Fanuc TP program (LS listing): both_features.ls

/PROG  BOTH_TEST
/ATTR
OWNER		= MNEDITOR;
COMMENT		= "";
PROG_SIZE	= 0;
CREATE		= DATE 24-01-23  TIME 05:57:44;
MODIFIED	= DATE 24-01-01  TIME 00:00:00;
FILE_NAME	= ;
VERSION		= 0;
LINE_COUNT	= 0;
MEMORY_SIZE	= 0;
PROTECT		= READ_WRITE;
TCD:  STACK_SIZE	= 0,
      TASK_PRIORITY	= 50,
      TIME_SLICE	= 0,
      BUSY_LAMP_OFF	= 0,
      ABORT_REQUEST	= 0,
      PAUSE_REQUEST	= 0;
DEFAULT_GROUP	= 1,*,*,*,*;
CONTROL_CODE	= 00000000 00000000;
/APPL
/MN
   :  R[1]=5 ;
   :  CALL MYPROG ;
   :   ;
/POS
/END
